FUNCTION_BLOCK TcoDoorCircuit EXTENDS TcoCore.TcoObject IMPLEMENTS ITcoDoorCircuit
VAR_INPUT
END_VAR
VAR_OUTPUT
END_VAR
VAR
	
	{attribute addProperty Name "<#Status#>"}
    {attribute clr [ReadOnly()]}
    _status : TcoDoorCircuit_Status;

	{attribute addProperty Name "<#Config#>"}
    _config : TcoDoorCircuit_Config;

	
	{attribute clr [RenderIgnore()]}
	_doors              : ARRAY [0..12] OF ITcoDoorLock;
		

	
	{attribute clr [RenderIgnore()]}
	_localDoorsVoltage  : ARRAY [0..4] OF ITcoControlVoltage;
	
	{attribute clr [RenderIgnore()]}
	_localVoltage  : ARRAY [0..4] OF ITcoControlVoltage;
	
	{attribute clr [RenderIgnore()]}
	_globalVoltage : ARRAY [0..4] OF ITcoControlVoltage;
	
	
	
    {attribute addProperty Name "<#Closed#>"}
    _isClosed : BOOL;
    
    {attribute addProperty Name "<#Locked#>"}
    _isLocked : BOOL;
    
    {attribute addProperty Name "<#Unlocked#>"}
    _isUnLocked : BOOL;
    
    {attribute addProperty Name "<#Global votage#>"}
    _isGlobalVoltageOk : BOOL;
    
    {attribute addProperty Name "<#Local voltage#>"}
    _isLocalVoltageOk : BOOL;
    
	 {attribute addProperty Name "<#Local Doors#>"}
    _isLocalDoorsVoltageOk : BOOL;


END_VAR

Initialize();

METHOD AddDoors : BOOL
VAR_INPUT
	inDoor : ITcoDoorLock;
END_VAR
VAR
	i : UINT;
END_VAR
AddDoors := FALSE;
FOR i := 0 TO _config.MaxDoors DO
	IF _doors[i] = inDoor THEN
		AddDoors := TRUE;
		RETURN;
	END_IF
	
	IF _doors[i] = 0 THEN
		_doors[i] := inDoor;
		AddDoors := TRUE;
		RETURN;
	END_IF
END_FOR
END_METHOD

METHOD AddGlobalVoltage : BOOL
VAR_INPUT
 	inVoltage : ITcoControlVoltage;
END_VAR
VAR
	i : UINT;
END_VAR
AddGlobalVoltage := FALSE;

IF inVoltage = 0 THEN
	RETURN;
END_IF

FOR i := 0 TO _config.MaxGlobalVoltage DO
	IF _globalVoltage[i] = inVoltage THEN
		addGlobalVoltage := TRUE;
		RETURN;
	END_IF
	
	IF 	_globalVoltage[i] = 0 THEN
		_globalVoltage[i] := inVoltage;
		addGlobalVoltage    := TRUE;
		RETURN;
	END_IF
END_FOR
END_METHOD

METHOD AddLocalDoorsVoltage : BOOL
VAR_INPUT
 	inVoltage : ITcoControlVoltage;
END_VAR
VAR
	i : UINT;
END_VAR
AddLocalDoorsVoltage := FALSE;

IF inVoltage = 0 THEN
	RETURN;
END_IF

FOR i := 0 TO _config.MaxLocalVoltage DO
	IF _localDoorsVoltage[i] = inVoltage THEN
		AddLocalDoorsVoltage := TRUE;
		RETURN;
	END_IF
	
	IF 	_localDoorsVoltage[i] = 0 THEN
		_localDoorsVoltage[i] := inVoltage;
		AddLocalDoorsVoltage    := TRUE;
		RETURN;
	END_IF
END_FOR
END_METHOD

METHOD AddLocalVoltage : BOOL
VAR_INPUT
 	inVoltage : ITcoControlVoltage;
END_VAR
VAR
	i : UINT;
END_VAR
addLocalVoltage := FALSE;

IF inVoltage = 0 THEN
	RETURN;
END_IF

FOR i := 0 TO _config.MaxLocalVoltage DO
	IF _localVoltage[i] = inVoltage THEN
		addLocalVoltage := TRUE;
		RETURN;
	END_IF
	
	IF 	_localVoltage[i] = 0 THEN
		_localVoltage[i] := inVoltage;
		addLocalVoltage    := TRUE;
		RETURN;
	END_IF
END_FOR
END_METHOD

PROPERTY Config :REFERENCE TO TcoDoorCircuit_Config
GET
Config ref=_config;
END_GET
END_PROPERTY

METHOD Initialize : BOOL
VAR
	d       : UINT;
	gv      : UINT;
	lv      : UINT;
	ldoors      : UINT;
	setOnce : BOOL;
END_VAR
// ------------------------------------------------------------- 
// 						GLOBAL VOLTAGE
// ------------------------------------------------------------- 
_isGlobalVoltageOk := FALSE;
setOnce            := FALSE;

FOR gv := 0 TO _config.MaxGlobalVoltage DO
	IF _globalVoltage[gv] <> 0 THEN
		IF NOT setOnce THEN
			_isGlobalVoltageOk := TRUE;
			setOnce := TRUE;
		END_IF
		
		IF _globalVoltage[gv].IsOff THEN
			_isGlobalVoltageOk := FALSE;
			EXIT;
		END_IF
	ELSE
		EXIT;
	END_IF
END_FOR

// ------------------------------------------------------------- 
// 						LOCAL VOLTAGE
// ------------------------------------------------------------- 
_isLocalVoltageOk := FALSE;
setOnce           := FALSE;

FOR lv := 0 TO _config.MaxLocalVoltage DO
	IF _localVoltage[lv] <> 0 THEN
		IF NOT setOnce THEN
			_isLocalVoltageOk := TRUE;
			setOnce := TRUE;
		END_IF
		
		IF _localVoltage[lv].IsOff THEN
			_isLocalVoltageOk := false;
			EXIT;
		END_IF
	ELSE
		EXIT;
	END_IF
END_FOR

// ------------------------------------------------------------- 
// 						LOCAL DOORS VOLTAGE OK
// ------------------------------------------------------------- 
_isLocalDoorsVoltageOk := FALSE;
setOnce           := FALSE;

FOR ldoors := 0 TO _config.MaxLocalDoorsVoltage DO
	IF _localDoorsVoltage[ldoors] <> 0 THEN
		IF NOT setOnce THEN
			_isLocalDoorsVoltageOk := TRUE;
			setOnce := TRUE;
		END_IF
		
		IF _localDoorsVoltage[ldoors].IsOff THEN
			_isLocalDoorsVoltageOk := FALSE;
			EXIT;
		END_IF
	ELSE
		EXIT;
	END_IF
END_FOR

// ------------------------------------------------------------- 
// 							DOORS
// ------------------------------------------------------------- 
_isClosed      := FALSE;
_isLocked      := FALSE;
_isUnLocked    := FALSE;
setOnce        := FALSE;
FOR d := 0 TO _config.MaxDoors DO
	IF _doors[d] <> 0 THEN
		IF NOT setOnce THEN
			setOnce        := TRUE;
			_isClosed      := TRUE;
			_isLocked      := TRUE;
			_isUnLocked    := TRUE;
		END_IF

		// Return TRUE only if all doors are Closed
		_isClosed   := _isClosed AND (_doors[d].IsClosed); // OR _doors[d].Deactivate);
		// Return TRUE only if all doors are Locked
		_isLocked   := _isLocked AND (_doors[d].IsLocked); //OR _doors[d].Deactivate);
		// Return TRUE only if all doors are Unlocked
		_isUnLocked := _isUnLocked AND NOT _doors[d].IsLocked;

	ELSE
		EXIT;
	END_IF
END_FOR
END_METHOD

{attribute 'monitoring' := 'variable'}
PROPERTY IsClosed : BOOL
GET
VAR
	d : UINT;
	setOnce : BOOL;
END_VAR
IsClosed := _isClosed ;
END_GET
END_PROPERTY

{attribute 'monitoring' := 'variable'}
PROPERTY IsGlobalVoltageOk : BOOL
GET
VAR
	gv : UINT;
END_VAR
IsGlobalVoltageOk := _isGlobalVoltageOk;
END_GET
END_PROPERTY

{attribute 'monitoring' := 'variable'}
PROPERTY IsLocalDoorsVoltageOk : BOOL
GET
VAR
	lv : UINT;
END_VAR
IsLocalDoorsVoltageOk := _isLocalDoorsVoltageOk;
END_GET
END_PROPERTY

{attribute 'monitoring' := 'variable'}
PROPERTY IsLocalVoltageOk : BOOL
GET
VAR
	lv : UINT;
END_VAR
IsLocalVoltageOk := _isLocalVoltageOk;
END_GET
END_PROPERTY

{attribute 'monitoring' := 'variable'}
PROPERTY IsLocked : BOOL
GET
VAR
	d : UINT;
	setOnce : BOOL;
END_VAR
IsLocked := _isLocked ;
END_GET
END_PROPERTY

{attribute 'monitoring' := 'variable'}
PROPERTY IsUnLocked : BOOL
GET
VAR
	d : UINT;
	setOnce : BOOL;
END_VAR
IsUnLocked := _isUnLocked;
END_GET
END_PROPERTY

METHOD Lock : BOOL
VAR_INPUT
END_VAR
VAR
	d : UINT;
END_VAR
Lock := FALSE;

IF NOT IsClosed THEN
	// we can't lock doors which are not closed
	RETURN;
END_IF

FOR d := 0 TO _config.MaxDoors DO
	IF _doors[d] <> 0 THEN
			_doors[d].Lock();
	ELSE
		EXIT;
	END_IF
END_FOR

Lock := THIS^.IsLocked;
END_METHOD

METHOD RemoveAllDoors
VAR
	i : UINT;
END_VAR
FOR i := 0 TO _config.MaxDoors DO
	_doors[i] := 0;
END_FOR
END_METHOD

METHOD RemoveDoors : BOOL
VAR_INPUT
	inDoorLock : ITcoDoorLock;
END_VAR
VAR
	i : UINT;
END_VAR
RemoveDoors := FALSE;

FOR i := 0 TO _config.MaxDoors DO 
	IF _doors[i] = inDoorLock THEN
		_doors[i] := 0;
		RemoveDoors :=  TRUE;
		RETURN;
	END_IF
END_FOR
END_METHOD

(*~
	<docu>
		<summary>
			Restores this instance to the Ready state. Can be called explicitly or from within one of the restore mechanisms.	
		</summary>			
	</docu>	
~*)
METHOD  Restore : ITcoRestorable

VAR
	i : UINT;
END_VAR
RemoveAllDoors();

FOR i := 0 TO _config.MaxGlobalVoltage DO
	_globalVoltage[i] := 0;
END_FOR

FOR i := 0 TO _config.MaxLocalVoltage DO
	_localVoltage[i] := 0;
END_FOR
FOR i := 0 TO _config.MaxLocalDoorsVoltage DO
	_localDoorsVoltage[i] := 0;
END_FOR
END_METHOD

(*~
	<docu>
		<summary>
		    Custom service (manual, maintenance) logic.
			This method must be implemented in derived class.
		</summary>			
	</docu>	
~*)
METHOD PROTECTED  ServiceMode
END_METHOD

PROPERTY Status : REFERENCE TO TcoDoorCircuit_Status
GET
Status REF=_status;
END_GET
END_PROPERTY

METHOD UnLock : BOOL
VAR
	d 		: UINT;
	setOnce : BOOL;
END_VAR
UnLock := FALSE;

FOR d := 0 TO _config.MaxDoors DO
	IF _doors[d] <> 0 THEN
		_doors[d].Unlock();
	ELSE
		exit;
	END_IF
END_FOR


FOR d := 0 TO _config.MaxDoors DO
	IF _doors[d] <> 0 THEN
		IF NOT setOnce THEN
			setOnce := TRUE;
			UnLock := TRUE;
		END_IF
		
		// return TRUE only if all doors are unlocked
		UnLock := Unlock AND NOT _doors[d].IsLocked;
	ELSE
		EXIT;
	END_IF
END_FOR
END_METHOD

END_FUNCTION_BLOCK

(* stored: Version 1.1.0.1
   POU TcoDoorCircuit: Id {73082c89-b7a7-4202-b3e8-7a6b095baf55}, SpecialFunc None
   Method AddDoors: Id {67485f30-a42f-4851-ad0e-22da5e378194}
   Method AddGlobalVoltage: Id {ccb8c6c6-0ed0-4992-99d4-6666ea63673e}
   Method AddLocalDoorsVoltage: Id {a0ac8e3f-a72a-49ce-a2ea-058ee1e8fa9a}
   Method AddLocalVoltage: Id {4e3e2766-414e-43a1-8fea-517e18bdf8db}
   Property Config: Id {2354fca6-11a8-4a80-bfd7-5d275e2c45c4}
   Get Get: Id {8868207c-1d0d-4d60-9426-b9a71364972b}
   Method Initialize: Id {b35c3fff-a359-4b4b-afe7-38d483a48be4}
   Property IsClosed: Id {af5ea3a0-6bdf-41e8-b234-9a560d2305c7}
   Get Get: Id {ebf6967f-9be8-45ec-aa6b-4f792a1f0a88}
   Property IsGlobalVoltageOk: Id {8dc91d3e-27fc-4fe8-b81e-57bf452b6915}
   Get Get: Id {ca0ae814-6622-41c9-8543-d00515f8e430}
   Property IsLocalDoorsVoltageOk: Id {4dca19b6-a34b-4cd9-9d04-d68853019a4b}
   Get Get: Id {5c44c4c5-391a-4b61-ba9a-8122ee61ef68}
   Property IsLocalVoltageOk: Id {7b8b3723-4c76-40aa-a81b-26c12135098c}
   Get Get: Id {9a6da6a8-2c49-4b0e-9ccc-358395e1ebfb}
   Property IsLocked: Id {2f01f034-a5af-4b86-8185-d2721deca0ed}
   Get Get: Id {7e99ac68-193d-420f-a1f3-9bfe6df4a29a}
   Property IsUnLocked: Id {dce07779-bd74-417a-a6c5-74258d0dd7f4}
   Get Get: Id {7d2fb05b-aa6e-458e-a2fb-0fd06f5a6b0c}
   Method Lock: Id {61208692-0229-473b-8970-2d35c6092bb2}
   Method RemoveAllDoors: Id {34f695cb-e2b9-4cf2-b03d-b8415b441716}
   Method RemoveDoors: Id {d06bb510-4db5-424e-8db0-a54b5ff58bb8}
   Method Restore: Id {9025b3de-8592-4d44-8702-498cf7e44e34}
   Method ServiceMode: Id {4b42fc2c-5f85-433e-9f4a-f151ee84d0c9}
   Property Status: Id {b5359157-c674-43e2-ae3a-3ae512b9af00}
   Get Get: Id {496830e9-4b54-4761-8e5e-6963207e1bc3}
   Method UnLock: Id {e9b12ab1-7993-48d3-97e3-deb4e96a6ef6} *)
